// TIA Portal project "Dynamic Setpoint Profiles" (V16)

(* hardware
DEVICE "S7-1200 station_1"  S7-1200 Station
   slot 0: "Rack_0"  S7-1200 Rack  Rack  V1.0
   slot 1: "PLC_1"  CPU 1212C DC/DC/DC  6ES7 212-1AE40-0XB0  V4.4
*)

// ===== PLC "PLC_1"  CPU 1212C DC/DC/DC =====

DATA_BLOCK "FB_TempRamp_Gen_DB"   // DB1
{ S7_Optimized_Access := 'TRUE' }
VERSION : 0.1
// stored: InstanceOfName FB_TempRamp_Gen
"FB_TempRamp_Gen"
BEGIN
END_DATA_BLOCK

FUNCTION_BLOCK "FB_TempRamp_Gen"   // FB1, SCL
{ S7_Optimized_Access := 'TRUE' }
VERSION : 0.1
   VAR_INPUT
      Start_Temp : Real;
      Target_Temp : Real;
      Ramp_Time_Min : Real;
      Enable : Bool;
      Reset : Bool;
      dt_sec : Real;
   END_VAR
   VAR_OUTPUT
      Output_Value : Real;
      Ramp_Complete : Bool;
   END_VAR
   VAR
      Elapsed_Time_sec : Real;
      Ramp_Rate : Real;
   END_VAR
BEGIN
   // 1. Calculate the rate of change in degrees per second

   IF #Ramp_Time_Min > 0.0 THEN
       #Ramp_Rate := (#Target_Temp - #Start_Temp) / (#Ramp_Time_Min * 60);
   ELSE
       #Ramp_Rate := 0.0;
   END_IF;

   // 2. Execution Logic
   IF #Reset THEN
       #Elapsed_Time_sec := 0.0;
       #Output_Value := #Start_Temp;
       #Ramp_Complete := FALSE;
   ELSIF #Enable AND NOT #Ramp_Complete THEN
       //// Accumulate elapsed time based on the execution cycle interval (dt)
       #Elapsed_Time_sec := #Elapsed_Time_sec + #dt_sec;
       // calculate the dynamic setpoint 
       #Output_Value := #Start_Temp + (#Ramp_Rate * #Elapsed_Time_sec);
       // 3. Failsafe Clamping and Completion Check for both Heating and Cooling
       IF (#Target_Temp >= #Start_Temp AND #Output_Value >= #Target_Temp)
           OR (#Target_Temp < #Start_Temp AND #Output_Value <= #Target_Temp) OR
           (#Ramp_Time_Min <= 0.0)THEN 
           #Output_Value := #Target_Temp;
           #Ramp_Complete := TRUE;
       END_IF;
   END_IF;
END_FUNCTION_BLOCK

ORGANIZATION_BLOCK "Main"   // OB1, LAD, ProgramCycle
TITLE = "Main Program Sweep (Cycle)"
{ S7_Optimized_Access := 'TRUE' }
VERSION : 0.1
   VAR_INPUT
      Initial_Call : Bool;   // Initial call of this OB
      Remanence : Bool;   // =True, if remanent data are available
   END_VAR
BEGIN
END_ORGANIZATION_BLOCK

ORGANIZATION_BLOCK "Cyclic interrupt"   // OB30, LAD, CyclicInterrupt
{ S7_Optimized_Access := 'TRUE' }
VERSION : 0.1
   VAR_INPUT
      Initial_Call : Bool;   // Initial call of this OB
      Event_Count : Int;   // Events discarded
   END_VAR
BEGIN

REGION Network 1
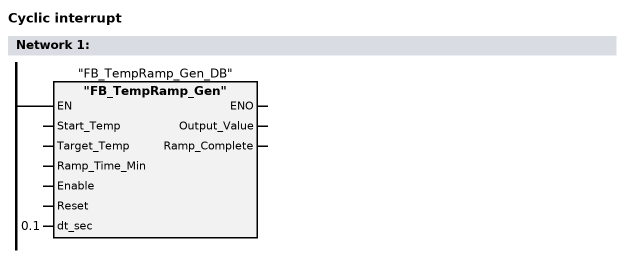
   RUNG wire#powerrail
      "FB_TempRamp_Gen_DB"(Start_Temp :=, Target_Temp :=, Ramp_Time_Min :=, Enable :=, Reset :=, dt_sec := 0.1, Output_Value =>, Ramp_Complete =>)
   END_RUNG
   // the same network as SCL:
   "FB_TempRamp_Gen_DB"(dt_sec := 0.1);   // "FB_TempRamp_Gen"
END_REGION
END_ORGANIZATION_BLOCK